INTERFACE I_NodeExecuteBeginEvent EXTENDS I_Event

PROPERTY PUBLIC Target : I_Node
GET
END_GET
END_PROPERTY

END_INTERFACE

(* stored: Version 1.1.0.1, ProductVersion 3.1.4024.12
   Itf I_NodeExecuteBeginEvent: Id {bf42bf61-5858-4802-b0c4-2b98bed0b96c}
   Property Target: Id {1552a38c-b4b5-4dc1-88ca-319e144ef719}
   Get Get: Id {bb5d5f4d-b0f6-41ed-a4f5-df5634ea05d2} *)
